(* CoDeSys 2.3 export: ENUMDALISENSOR.EXP *)

(* Data type *)
TYPE enumDaliSensor :
(
	NoSensor := 0, (* default type is no sensor *)
	MultiSensorType1,
	PushbuttonSensorType1,
	MultiSensorType2,
	PushbuttonSensorType2,
	DaliEcg,
	DaliGroup
);
END_TYPE
